TYPE IData :
STRUCT
	strBetryName:STRING;//CCD给电芯名称 
	bNGOverHang :BOOL;  //
	bHaveBetry :BOOL;   //当前工位是否有电芯
    
	
	bNGShort:BOOL;  //短路NG
	strShortData:STRING; //短路测试数据
	
	strCode:STRING;//二维码
    bNGCode:BOOL;   //二维码NG
	
	strHotPress:STRING;//热压参数
END_STRUCT
END_TYPE

(* stored: Version 1.1.0.1, ProductVersion 3.1.4024.9
   DUT IData: Id {008cac40-a37f-406f-93e5-f9a13fd71ea5} *)
